// TIA Portal V21 export
TYPE "switchgearStopCtx"
   STRUCT
      "step" : USInt;
      stepTime : LTime;
      alm : "switchgearAlm";
      almWord { S7_SetPoint := 'True'} : Word;
   END_STRUCT;
END_TYPE
